{attribute 'qualified_only'}
VAR_GLOBAL CONSTANT
	
	// JBOX TESTER CONSTANTS
	HMI_HOME_NUM_INSTRUCTIONS : INT := 8;
	HMI_SECTION_1_NUM_INSTRUCTIONS : INT := 7;
	HMI_SECTION_2_NUM_INSTRUCTIONS : INT := 8;
	TOTAL_NUM_TESTS : INT := 70;
	SECTION1_NUM_DIG_TESTS : INT := 24;
	SECTION1_NUM_HMI_TESTS : INT := 4;
	SECTION2_NUM_DIG_TESTS : INT := 19;
	SECTION2_NUM_HMI_TESTS : INT := 3;
	NUM_CONNECTIONS : INT := 28;
	
	
END_VAR

(* stored: Version 1.1.0.1, ProductVersion 3.1.4024.10
   GVL CONSTANTS: Id {971eb940-d70a-4e58-93b7-490745d09d4e}, ParameterList True *)
